// TIA Portal V18 export
TYPE "PLCtoMES_ProcessingExchange"
// stored: IsFailsafeCompliant false
   STRUCT
      "P-ProcessingPartID" : String[48];   // P-Processing置位和复位期间需要保持这个ID数据
      "P-ProcessingReq" : Bool;   // 不可逆加工状态位，当此信号只有上升沿没有下降沿，MES标记此工件ID为不可二次加工并判断该产品为PartNG.
      Reserve : Array[1..248] of Byte;   // SubPartReq子零件绑定交互预留
   END_STRUCT;
END_TYPE
